(* IEC 61131-3 sources: inj-machine-docs/docs/IM_SYS_PRG/Code/面板管理, 4 files *)

(* ---- PanelTypes.st ---- *)
(*
  PanelTypes.st
  功能：
  1. 定义面板管理层统一使用的按键点位结构和综合按键结构。
  2. 统一收口“面板排序号 + 按键值 + 按键灯”三类信息，避免键值与灯值分散绑定。
  3. 为 `FB_MK110`、`FB_MK116`、`FB_MK150` 提供稳定的数据边界。

  说明：
  1. `uiPanelOrder` 由具体面板功能块按各自型号写入，`0` 表示当前面板未安装该逻辑键位。
  2. `bValue` 由面板输入解码逻辑回写，表示当前逻辑键是否被按下。
  3. `bLamp` 由上层控制逻辑写入，表示当前逻辑键对应的灯是否需要点亮。
*)

TYPE ST_PanelButton :
STRUCT
    uiPanelOrder: UINT;     // 当前逻辑键在当前面板型号中的排序号；`0` 表示该面板型号不提供此键位。
    bValue: BOOL;           // 当前逻辑键输入值；由面板功能块根据输入字和排序号解码后回写。
    bLamp: BOOL;            // 当前逻辑键灯输出请求；由上层写入，再由面板功能块按排序号编码到输出字。
END_STRUCT
END_TYPE

TYPE ST_PanelButtons :
STRUCT
    stManual: ST_PanelButton;            // 手动键综合点位，统一收口其排序号、键值和灯值。
    stSemiautomatic: ST_PanelButton;     // 半自动键综合点位，统一收口其排序号、键值和灯值。
    stAutomatic: ST_PanelButton;         // 全自动键综合点位，统一收口其排序号、键值和灯值。
    stAdjustMold: ST_PanelButton;        // 调模键综合点位，统一收口其排序号、键值和灯值。
    stHeat: ST_PanelButton;              // 电热键综合点位，统一收口其排序号、键值和灯值。
    stMotor: ST_PanelButton;             // 马达键综合点位，统一收口其排序号、键值和灯值。
    stMoldOpen: ST_PanelButton;          // 开模键综合点位，统一收口其排序号、键值和灯值。
    stMoldClose: ST_PanelButton;         // 锁模键综合点位，统一收口其排序号、键值和灯值。
    stMaterialMelt: ST_PanelButton;      // 储料键综合点位，统一收口其排序号、键值和灯值。
    stCleanMaterial: ST_PanelButton;     // 清料键综合点位，统一收口其排序号、键值和灯值。
    stJetLube: ST_PanelButton;           // 润滑键综合点位，统一收口其排序号、键值和灯值。
    stInjFwd: ST_PanelButton;            // 射出键综合点位，统一收口其排序号、键值和灯值。
    stInjBwd: ST_PanelButton;            // 射退键综合点位，统一收口其排序号、键值和灯值。
    stZipperBwd: ST_PanelButton;         // 倒带键综合点位，统一收口其排序号、键值和灯值。
    stZipperFwd: ST_PanelButton;         // 拉带键综合点位，统一收口其排序号、键值和灯值。
    stPressRise: ST_PanelButton;         // 压力加键综合点位，统一收口其排序号、键值和灯值。
    stPressFall: ST_PanelButton;         // 压力减键综合点位，统一收口其排序号、键值和灯值。
    stEjectorFwd: ST_PanelButton;        // 托模进键综合点位，统一收口其排序号、键值和灯值。
    stEjectorBwd: ST_PanelButton;        // 托模退键综合点位，统一收口其排序号、键值和灯值。
    stMultiEjector: ST_PanelButton;      // 多次托模键综合点位，统一收口其排序号、键值和灯值。
    stBlow: ST_PanelButton;              // 吹气键综合点位，统一收口其排序号、键值和灯值。
    stZipperClamp: ST_PanelButton;       // 夹带键综合点位，统一收口其排序号、键值和灯值。
    stZipperMotor: ST_PanelButton;       // 拉带马达键综合点位，统一收口其排序号、键值和灯值。
    stInjUnitFwd: ST_PanelButton;        // 座进键综合点位，统一收口其排序号、键值和灯值。
    stInjUnitBwd: ST_PanelButton;        // 座退键综合点位，统一收口其排序号、键值和灯值。
    stLockFwd: ST_PanelButton;           // 定位进键综合点位，统一收口其排序号、键值和灯值。
    stLockBwd: ST_PanelButton;           // 定位退键综合点位，统一收口其排序号、键值和灯值。
    stCoreFwdA: ST_PanelButton;          // 中子 A 进键综合点位，统一收口其排序号、键值和灯值。
    stCoreBwdA: ST_PanelButton;          // 中子 A 退键综合点位，统一收口其排序号、键值和灯值。
END_STRUCT
END_TYPE

(* ---- F_PanelGetBit.st ---- *)
(*
  F_PanelGetBit 函数
  功能：
  1. 从一个 `WORD` 中按位索引读取单个布尔值。
  2. 供面板输入解码函数按“字 + 位”的方式统一读取按键输入。
  3. 越界位索引会直接返回 `FALSE`，避免上层再额外做边界保护。
*)
FUNCTION F_PanelGetBit : BOOL
VAR_INPUT
    wValue: WORD;          // 待读取的源字；通常来自面板输入字 `wIN0~wIN3`。
    uiBitIndex: UINT;      // 目标位索引；有效范围为 `0..15`。
END_VAR

IF uiBitIndex > 15 THEN
    F_PanelGetBit := FALSE;                                                        // 位索引越界时直接返回 FALSE，避免把非法位误判为有效输入。
ELSE
    F_PanelGetBit := ((SHR(wValue, uiBitIndex) AND WORD#1) = WORD#1);              // 位索引有效时，把目标位右移到最低位后判断其是否为 1。
END_IF;
END_FUNCTION

(* ---- F_PanelSetBit.st ---- *)
(*
  F_PanelSetBit 函数
  功能：
  1. 按位索引对一个 `WORD` 做置位或清位操作。
  2. 供面板灯输出逻辑按“排序号 -> 输出位”的方式统一生成输出字。
  3. 越界位索引会直接返回原字，避免上层输出字被非法写坏。
*)
FUNCTION F_PanelSetBit : WORD
VAR_INPUT
    wValue: WORD;          // 待修改的目标字；通常来自面板输出字 `wOUT0` 或 `wOUT1`。
    uiBitIndex: UINT;      // 目标位索引；有效范围为 `0..15`。
    bBitValue: BOOL;       // TRUE=把目标位置 1；FALSE=把目标位清 0。
END_VAR

IF uiBitIndex > 15 THEN
    F_PanelSetBit := wValue;                                                      // 位索引越界时保持原字不变，避免误改无关输出位。
ELSIF bBitValue THEN
    F_PanelSetBit := wValue OR SHL(WORD#1, uiBitIndex);                           // 需要点亮时，用位掩码把目标位置 1。
ELSE
    F_PanelSetBit := wValue AND NOT SHL(WORD#1, uiBitIndex);                      // 需要熄灭时，用位掩码把目标位清 0。
END_IF;
END_FUNCTION

(* ---- FB_PanelLampWriter.st ---- *)
(*
  FB_PanelLampWriter 功能块
  功能：
  1. 按统一的面板排序号，把单个逻辑键的灯请求写入 `wOUT0/wOUT1`。
  2. 约定排序号 `1..16` 对应 `wOUT0` 的 `0..15` 位，排序号 `17..32` 对应 `wOUT1` 的 `0..15` 位。
  3. 供 `FB_MK110`、`FB_MK116`、`FB_MK150` 复用，避免每个面板块重复展开灯位写入分支。

  使用约束：
  1. 调用方必须在本扫描周期开始前先把 `wOUT0`、`wOUT1` 清零。
  2. 本块只负责把单个逻辑键的灯请求并入输出字，不负责排序号唯一性检查。
*)
FUNCTION_BLOCK FB_PanelLampWriter
VAR_IN_OUT
    wOUT0: WORD;              // 输出字 0；承载排序号 `1..16` 对应的面板灯位。
    wOUT1: WORD;              // 输出字 1；承载排序号 `17..32` 对应的面板灯位。
END_VAR
VAR_INPUT
    uiPanelOrder: UINT;       // 当前逻辑键在当前面板型号中的排序号；`0` 表示本次不写任何灯位。
    bLampValue: BOOL;         // 当前逻辑键的灯请求；TRUE=点亮对应灯位，FALSE=保持输出字当前值不变。
END_VAR

IF NOT bLampValue THEN
    (* 当前逻辑键灯请求为 FALSE 时不做任何写入。
       调用方已在扫描周期开始时统一清零输出字，因此这里不需要再重复清位。
    *)
ELSIF (uiPanelOrder >= 1) AND (uiPanelOrder <= 16) THEN
    wOUT0 := F_PanelSetBit(wValue := wOUT0, uiBitIndex := uiPanelOrder - 1, bBitValue := TRUE);      // 排序号落在 `1..16` 时，把灯写入 `wOUT0` 的对应位。
ELSIF (uiPanelOrder >= 17) AND (uiPanelOrder <= 32) THEN
    wOUT1 := F_PanelSetBit(wValue := wOUT1, uiBitIndex := uiPanelOrder - 17, bBitValue := TRUE);     // 排序号落在 `17..32` 时，把灯写入 `wOUT1` 的对应位。
END_IF;
END_FUNCTION_BLOCK
